// TIA Portal V18 export
DATA_BLOCK "PARAMs"   // DB17
{ S7_Optimized_Access := 'TRUE' }
VERSION : 0.1
// stored: AutoNumber true, DBAccessibleFromOPCUA true, IsOnlyStoredInLoadMemory false, IsRetainMemResEnabled false, IsWriteProtectedInAS false, MemoryReserve 100
   VAR
      K_min_v : Real := 0.1;
      K_min_dist : Real := 0.003;
      K_dist_fast : Real := 5.0;
   END_VAR
   VAR RETAIN
      M1Z { S7_SetPoint := 'True'} : "typeMotPara";
      M2Y { S7_SetPoint := 'True'} : "typeMotPara";
      M3X { S7_SetPoint := 'True'} : "typeMotPara";
      M4O1 { S7_SetPoint := 'True'} : "typeMotPara";
      M5O2 { S7_SetPoint := 'True'} : "typeMotPara";
      M6Doors { S7_SetPoint := 'True'} : "typeMotPara";
   END_VAR
BEGIN
   M1Z.t_acc_50Hz_USER := 10.0;
   M1Z.v_absoluteMax_LOGIC := 113.3333;
   M1Z.dist_absMax_LOGIC := 581.6667;
   M1Z.v_crawl_USER := 3.0;
   M1Z.dist_crawl_USER := 3.0;
   M1Z.dist_stop_USER := 1.0;
   M1Z.dist_auto_done_LOGIC := 3.0;
   M1Z.pos_calib_USER := 0.0;
   M1Z.pos_lim_fwd_USER := 100.0;
   M1Z.pos_lim_rev_USER := 0.0;
   M1Z.v_blind_USER := 0.0;
   M1Z.v_manual_USER := 0.0;
   M1Z.v_auto_USER := 0.0;
   M1Z.t_er := T#1S;
   M2Y.t_acc_50Hz_USER := 10.0;
   M2Y.v_absoluteMax_LOGIC := 111.6667;
   M2Y.dist_absMax_LOGIC := 608.3333;
   M2Y.v_crawl_USER := 10.0;
   M2Y.dist_crawl_USER := 5.0;
   M2Y.dist_stop_USER := 1.0;
   M2Y.dist_auto_done_LOGIC := 3.0;
   M2Y.pos_calib_USER := 0.0;
   M2Y.pos_lim_fwd_USER := 847.0;
   M2Y.pos_lim_rev_USER := 0.0;
   M2Y.v_blind_USER := 20.0;
   M2Y.v_manual_USER := 50.0;
   M2Y.v_auto_USER := 60.0;
   M2Y.t_er := T#3S;
   M3X.t_acc_50Hz_USER := 3.0;
   M3X.v_absoluteMax_LOGIC := 118.3696;
   M3X.dist_absMax_LOGIC := 185.0543;
   M3X.v_crawl_USER := 5.0;
   M3X.dist_crawl_USER := 2.0;
   M3X.dist_stop_USER := 1.0;
   M3X.dist_auto_done_LOGIC := 3.0;
   M3X.pos_calib_USER := 0.0;
   M3X.pos_lim_fwd_USER := 680.0;
   M3X.pos_lim_rev_USER := 0.0;
   M3X.v_blind_USER := 10.0;
   M3X.v_manual_USER := 50.0;
   M3X.v_auto_USER := 100.0;
   M3X.t_er := T#3S;
   M4O1.t_acc_50Hz_USER := 1.0;
   M4O1.v_absoluteMax_LOGIC := 31.17822;
   M4O1.dist_absMax_LOGIC := 17.08911;
   M4O1.v_crawl_USER := 3.0;
   M4O1.dist_crawl_USER := 2.0;
   M4O1.dist_stop_USER := 1.0;
   M4O1.dist_auto_done_LOGIC := 3.0;
   M4O1.pos_calib_USER := 0.0;
   M4O1.pos_lim_fwd_USER := 5.0;
   M4O1.pos_lim_rev_USER := 0.0;
   M4O1.v_blind_USER := 3.0;
   M4O1.v_manual_USER := 3.0;
   M4O1.v_auto_USER := 1.0;
   M4O1.t_er := T#3S;
   M5O2.t_acc_50Hz_USER := 10.0;
   M5O2.v_absoluteMax_LOGIC := 67.0;
   M5O2.dist_absMax_LOGIC := 345.0;
   M5O2.v_crawl_USER := 2.0;
   M5O2.dist_crawl_USER := 2.0;
   M5O2.dist_stop_USER := 0.2;
   M5O2.dist_auto_done_LOGIC := 0.6;
   M5O2.pos_calib_USER := 0.0;
   M5O2.pos_lim_fwd_USER := 360.0;
   M5O2.pos_lim_rev_USER := 0.0;
   M5O2.v_blind_USER := 30.0;
   M5O2.v_manual_USER := 30.0;
   M5O2.v_auto_USER := 50.0;
   M5O2.t_er := T#3S;
   M6Doors.t_acc_50Hz_USER := 10.0;
   M6Doors.v_absoluteMax_LOGIC := 83.33334;
   M6Doors.dist_absMax_LOGIC := 446.6667;
   M6Doors.v_crawl_USER := 6.0;
   M6Doors.dist_crawl_USER := 6.0;
   M6Doors.dist_stop_USER := 3.0;
   M6Doors.dist_auto_done_LOGIC := 9.0;
   M6Doors.pos_calib_USER := 0.0;
   M6Doors.pos_lim_fwd_USER := 1.0;
   M6Doors.pos_lim_rev_USER := 0.0;
   M6Doors.v_blind_USER := 5.0;
   M6Doors.v_manual_USER := 5.0;
   M6Doors.v_auto_USER := 5.0;
   M6Doors.t_er := T#3S;
END_DATA_BLOCK
